{attribute addProperty BoxType "EL9540-0010-0016"}
{attribute addProperty Id "Status_UpAT %I*Status_Up_B12359DC1620WcStateAT %I*WcState_F855686C1620InfoDataAT %I*InfoData_192954DE1620"}
{attribute addProperty CRC "1308685549"}
{attribute addProperty SizeInBites "48"}
{attribute addProperty SizeInBytes "6"}
TYPE EL9540_7D2BCDCD :
STRUCT
	{attribute addProperty Name "Status_Up"}
	Status_Up : Status_Up_B12359DC;
	{attribute addProperty Name "WcState"}
	WcState : WcState_F855686C;
	{attribute addProperty Name "InfoData"}
	InfoData : InfoData_192954DE;
END_STRUCT
END_TYPE

(* stored: Version 1.2.0.0, ProductVersion 3.1.4024.9
   DUT EL9540_7D2BCDCD: Id {e561ebe4-1204-4940-95dd-1a8a4d000ff3} *)
